(* PLC project Recipe_Tool, Beckhoff Automation GmbH TwinCAT PLC Control 3.5.3.40 *)
(* stored: creationDateTime 2014-11-22T03:13:17.8029505, modificationDateTime 2014-11-22T03:13:17.8029505 *)

FUNCTION_BLOCK Recipe_10051_FreePassion
  VAR_INPUT
    execute : BOOL;
    Order : DUT_RECIPEORDER;
  END_VAR
  VAR_OUTPUT
    RecipeInfo : DUT_RECIPEOFFER;
    RecipeDone : BOOL;
    InitDone : BOOL;
  END_VAR
  VAR
    userparametersum : LREAL;
    StepDone : BOOL;
    i : INT;
  END_VAR

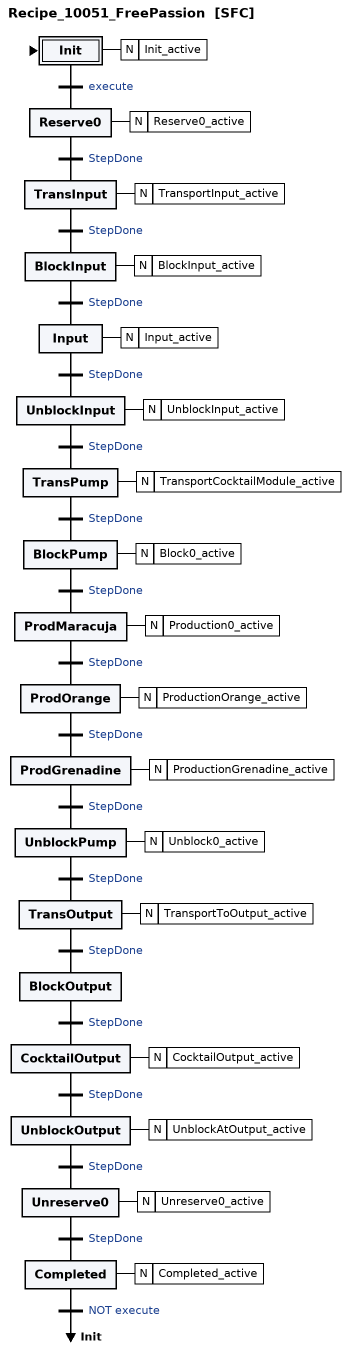
INITIAL_STEP Init:
  Init_active(N);
END_STEP
TRANSITION FROM Init TO Reserve0
  := execute;
END_TRANSITION
STEP Reserve0:
  Reserve0_active(N);
END_STEP
TRANSITION FROM Reserve0 TO TransInput
  := StepDone;
END_TRANSITION
STEP TransInput:
  TransportInput_active(N);
END_STEP
TRANSITION FROM TransInput TO BlockInput
  := StepDone;
END_TRANSITION
STEP BlockInput:
  BlockInput_active(N);
END_STEP
TRANSITION FROM BlockInput TO Input
  := StepDone;
END_TRANSITION
STEP Input:
  Input_active(N);
END_STEP
TRANSITION FROM Input TO UnblockInput
  := StepDone;
END_TRANSITION
STEP UnblockInput:
  UnblockInput_active(N);
END_STEP
TRANSITION FROM UnblockInput TO TransPump
  := StepDone;
END_TRANSITION
STEP TransPump:
  TransportCocktailModule_active(N);
END_STEP
TRANSITION FROM TransPump TO BlockPump
  := StepDone;
END_TRANSITION
STEP BlockPump:
  Block0_active(N);
END_STEP
TRANSITION FROM BlockPump TO ProdMaracuja
  := StepDone;
END_TRANSITION
STEP ProdMaracuja:
  Production0_active(N);
END_STEP
TRANSITION FROM ProdMaracuja TO ProdOrange
  := StepDone;
END_TRANSITION
STEP ProdOrange:
  ProductionOrange_active(N);
END_STEP
TRANSITION FROM ProdOrange TO ProdGrenadine
  := StepDone;
END_TRANSITION
STEP ProdGrenadine:
  ProductionGrenadine_active(N);
END_STEP
TRANSITION FROM ProdGrenadine TO UnblockPump
  := StepDone;
END_TRANSITION
STEP UnblockPump:
  Unblock0_active(N);
END_STEP
TRANSITION FROM UnblockPump TO TransOutput
  := StepDone;
END_TRANSITION
STEP TransOutput:
  TransportToOutput_active(N);
END_STEP
TRANSITION FROM TransOutput TO BlockOutput
  := StepDone;
END_TRANSITION
STEP BlockOutput:
END_STEP
TRANSITION FROM BlockOutput TO CocktailOutput
  := StepDone;
END_TRANSITION
STEP CocktailOutput:
  CocktailOutput_active(N);
END_STEP
TRANSITION FROM CocktailOutput TO UnblockOutput
  := StepDone;
END_TRANSITION
STEP UnblockOutput:
  UnblockAtOutput_active(N);
END_STEP
TRANSITION FROM UnblockOutput TO Unreserve0
  := StepDone;
END_TRANSITION
STEP Unreserve0:
  Unreserve0_active(N);
END_STEP
TRANSITION FROM Unreserve0 TO Completed
  := StepDone;
END_TRANSITION
STEP Completed:
  Completed_active(N);
END_STEP
TRANSITION FROM Completed TO Init
  := NOT execute;
END_TRANSITION

ACTION Completed_active:
                RecipeDone := TRUE;
StepDone := FALSE;
              
END_ACTION

ACTION Init_active:
                RecipeDone := FALSE;

// Initialisation of Recipe Parameters an name etc
RecipeInfo.Name := 'Free Passion';
RecipeInfo.Description := 'Sweet cocktail combining the sourness of Maracuja juice with the sweetness of grenadine syrup';
RecipeInfo.Dummy := FALSE;
RecipeInfo.RecipeID := 10051; 	// 
Initdone := TRUE;

//Parameter 0:

	RecipeInfo.UserParameter[0].Dummy 		:= FALSE
	RecipeInfo.UserParameter[0].Default		:= '200'
	RecipeInfo.UserParameter[0].Description	:= 'Gives the total fluid amount in the glass'
	RecipeInfo.UserParameter[0].MaxValue	:= 200
	RecipeInfo.UserParameter[0].MinValue	:= 10
	RecipeInfo.UserParameter[0].Name		:= 'Amount'
	RecipeInfo.UserParameter[0].Unit		:= 'ml'
	
//Parameter 1:

	RecipeInfo.UserParameter[1].Dummy 		:= FALSE
	RecipeInfo.UserParameter[1].Default		:= '50'
	RecipeInfo.UserParameter[1].Description	:= 'Maracuja Juice'
	RecipeInfo.UserParameter[1].MaxValue	:= 100
	RecipeInfo.UserParameter[1].MinValue	:= 1
	RecipeInfo.UserParameter[1].Name		:= 'Maracuja Juice'
	RecipeInfo.UserParameter[1].Unit		:= 'ml'
	
//Parameter 2:

	RecipeInfo.UserParameter[2].Dummy 		:= FALSE
	RecipeInfo.UserParameter[2].Default		:= '35'
	RecipeInfo.UserParameter[2].Description	:= 'Orange Juice'
	RecipeInfo.UserParameter[2].MaxValue	:= 100
	RecipeInfo.UserParameter[2].MinValue	:= 1
	RecipeInfo.UserParameter[2].Name		:= 'Orange Juice'
	RecipeInfo.UserParameter[2].Unit		:= 'ml'

//Parameter 3:

	RecipeInfo.UserParameter[3].Dummy 		:= FALSE
	RecipeInfo.UserParameter[3].Default		:= '15'
	RecipeInfo.UserParameter[3].Description	:= 'Grenadine Syrup'
	RecipeInfo.UserParameter[3].MaxValue	:= 50
	RecipeInfo.UserParameter[3].MinValue	:= 1
	RecipeInfo.UserParameter[3].Name		:= 'Grenadine Syrup'
	RecipeInfo.UserParameter[3].Unit		:= 'ml'
	
	
	
//Parameter 1:
(*
	RecipeInfo.UserParameter[1].Dummy 		:= 
	RecipeInfo.UserParameter[1].Default		:=
	RecipeInfo.UserParameter[1].Description	:=
	RecipeInfo.UserParameter[1].MaxValue	:=
	RecipeInfo.UserParameter[1].MinValue	:=
	RecipeInfo.UserParameter[1].Name		:=
	RecipeInfo.UserParameter[1].Unit		:=
*)
//Parameter 2:

(*
	RecipeInfo.UserParameter[2].Dummy 		:= 
	RecipeInfo.UserParameter[2].Default		:=
	RecipeInfo.UserParameter[2].Description	:=
	RecipeInfo.UserParameter[2].MaxValue	:=
	RecipeInfo.UserParameter[2].MinValue	:=
	RecipeInfo.UserParameter[2].Name		:=
	RecipeInfo.UserParameter[2].Unit		:=
*)

//Parameter 3:

(*
	RecipeInfo.UserParameter[3].Dummy 		:= 
	RecipeInfo.UserParameter[3].Default		:=
	RecipeInfo.UserParameter[3].Description	:=
	RecipeInfo.UserParameter[3].MaxValue	:=
	RecipeInfo.UserParameter[3].MinValue	:=
	RecipeInfo.UserParameter[3].Name		:=
	RecipeInfo.UserParameter[3].Unit		:=
*)

//Parameter 4:

(*
	RecipeInfo.UserParameter[4].Dummy 		:= 
	RecipeInfo.UserParameter[4].Default		:=
	RecipeInfo.UserParameter[4].Description	:=
	RecipeInfo.UserParameter[4].MaxValue	:=
	RecipeInfo.UserParameter[4].MinValue	:=
	RecipeInfo.UserParameter[4].Name		:=
	RecipeInfo.UserParameter[4].Unit		:=
*)


//Parameter 5:

(*
	RecipeInfo.UserParameter[5].Dummy 		:= 
	RecipeInfo.UserParameter[5].Default		:=
	RecipeInfo.UserParameter[5].Description	:=
	RecipeInfo.UserParameter[5].MaxValue	:=
	RecipeInfo.UserParameter[5].MinValue	:=
	RecipeInfo.UserParameter[5].Name		:=
	RecipeInfo.UserParameter[5].Unit		:=
*)
              
END_ACTION

ACTION Reserve0_active:
                StepDone := FALSE;
RecipeDone := FALSE;
//Skill auswählen
ExecuteSkill.SkillID 		:= 1310;
ExecuteSkill.SkillName	 	:= 'Reserve';

//Parameter setzen

ExecuteSkill.Parameter[1].ID := 1;
ExecuteSkill.Parameter[1].Name := 'TaskID';
ExecuteSkill.Parameter[1].Value := Order.TaskID;


(*
ExecuteSkill.Parameter[2].ID := ;
ExecuteSkill.Parameter[2].Name := '';
ExecuteSkill.Parameter[2].Value := ;
*)

(*
ExecuteSkill.Parameter[3].ID := ;
ExecuteSkill.Parameter[3].Name := '';
ExecuteSkill.Parameter[3].Value := ;
*)

(*
ExecuteSkill.Parameter[4].ID := ;
ExecuteSkill.Parameter[4].Name := '';
ExecuteSkill.Parameter[4].Value := ;
*)

(*
ExecuteSkill.Parameter[5].ID := ;
ExecuteSkill.Parameter[5].Name := '';
ExecuteSkill.Parameter[5].Value := ;
*)



ExecuteSkill();

StepDone := ExecuteSkill.Done;
              
END_ACTION

ACTION Production0_active:
                StepDone := FALSE;

userparametersum := 0;
FOR i := 1 TO UserParameterCnt DO
	IF NOT order.UserParameter[i].Value = 0 THEN
		userparametersum := userparametersum + order.UserParameter[i].Value;
	END_IF
END_FOR
//Skill auswählen
ExecuteSkill.SkillID 		:= 1113;
ExecuteSkill.SkillName	 	:= 'Marajuca Juice';

//Parameter setzen

ExecuteSkill.Parameter[1].ID := 1;
ExecuteSkill.Parameter[1].Name := 'Quantity';
//order.userParameter[0] = amount
ExecuteSkill.Parameter[1].Value := order.UserParameter[0].Value * order.UserParameter[0].Value / userparametersum;//Summe aller Zutatenmengen;


(*
ExecuteSkill.Parameter[2].ID := ;
ExecuteSkill.Parameter[2].Name := '';
ExecuteSkill.Parameter[2].Value := ;
*)

(*
ExecuteSkill.Parameter[3].ID := ;
ExecuteSkill.Parameter[3].Name := '';
ExecuteSkill.Parameter[3].Value := ;
*)

(*
ExecuteSkill.Parameter[4].ID := ;
ExecuteSkill.Parameter[4].Name := '';
ExecuteSkill.Parameter[4].Value := ;
*)

(*
ExecuteSkill.Parameter[5].ID := ;
ExecuteSkill.Parameter[5].Name := '';
ExecuteSkill.Parameter[5].Value := ;
*)



ExecuteSkill();

StepDone := ExecuteSkill.Done;
              
END_ACTION

ACTION ProductionOrange_active:
                StepDone := FALSE;

//Skill auswählen
ExecuteSkill.SkillID 		:= 1117;
ExecuteSkill.SkillName	 	:= 'Orange';

//Parameter setzen

ExecuteSkill.Parameter[1].ID := 1;
ExecuteSkill.Parameter[1].Name := 'Quantity';
//order.userParameter[0] = amount
ExecuteSkill.Parameter[1].Value := order.UserParameter[0].Value * order.UserParameter[1].Value / userparametersum;//Summe aller Zutatenmengen;



(*
ExecuteSkill.Parameter[2].ID := ;
ExecuteSkill.Parameter[2].Name := '';
ExecuteSkill.Parameter[2].Value := ;
*)

(*
ExecuteSkill.Parameter[3].ID := ;
ExecuteSkill.Parameter[3].Name := '';
ExecuteSkill.Parameter[3].Value := ;
*)

(*
ExecuteSkill.Parameter[4].ID := ;
ExecuteSkill.Parameter[4].Name := '';
ExecuteSkill.Parameter[4].Value := ;
*)

(*
ExecuteSkill.Parameter[5].ID := ;
ExecuteSkill.Parameter[5].Name := '';
ExecuteSkill.Parameter[5].Value := ;
*)



ExecuteSkill();

StepDone := ExecuteSkill.Done;
              
END_ACTION

ACTION ProductionGrenadine_active:
                StepDone := FALSE;

//Skill auswählen
ExecuteSkill.SkillID 		:= 1111;
ExecuteSkill.SkillName	 	:= 'Grenadine';

//Parameter setzen

ExecuteSkill.Parameter[1].ID := 1;
ExecuteSkill.Parameter[1].Name := 'Quantity';
//order.userParameter[0] = amount
ExecuteSkill.Parameter[1].Value := order.UserParameter[0].Value * order.UserParameter[2].Value / userparametersum; //Summe aller Zutatenmengen;



(*
ExecuteSkill.Parameter[2].ID := ;
ExecuteSkill.Parameter[2].Name := '';
ExecuteSkill.Parameter[2].Value := ;
*)

(*
ExecuteSkill.Parameter[3].ID := ;
ExecuteSkill.Parameter[3].Name := '';
ExecuteSkill.Parameter[3].Value := ;
*)

(*
ExecuteSkill.Parameter[4].ID := ;
ExecuteSkill.Parameter[4].Name := '';
ExecuteSkill.Parameter[4].Value := ;
*)

(*
ExecuteSkill.Parameter[5].ID := ;
ExecuteSkill.Parameter[5].Name := '';
ExecuteSkill.Parameter[5].Value := ;
*)



ExecuteSkill();

StepDone := ExecuteSkill.Done;
              
END_ACTION

ACTION TransportCocktailModule_active:
                StepDone := FALSE;

//Skill auswählen
ExecuteSkill.SkillID 		:= 1320;
ExecuteSkill.SkillName	 	:= 'Transport';

//Parameter setzen

ExecuteSkill.Parameter[3].ID := 3;
ExecuteSkill.Parameter[3].Name := 'Velocity';
ExecuteSkill.Parameter[3].Value := 300;



ExecuteSkill.Parameter[1].ID :=  1;
ExecuteSkill.Parameter[1].Name := 'TargetPosition X';
ExecuteSkill.Parameter[1].Value := 30 ;
ExecuteSkill.Parameter[1].StringValue := '#DP#2#XPosition';



ExecuteSkill.Parameter[2].ID := 2;
ExecuteSkill.Parameter[2].Name := 'TargetPosition Z';
ExecuteSkill.Parameter[2].Value := 10;// ZCookieModule - ZCookieModuleCalibration - 2* Cookiethickness + toppingthickness+ Preasureheight  ;



(*
ExecuteSkill.Parameter[4].ID := 4;
ExecuteSkill.Parameter[4].Name := 'Acceleration';
ExecuteSkill.Parameter[4].Value := 0 ;
*)

(*
ExecuteSkill.Parameter[5].ID := ;
ExecuteSkill.Parameter[5].Name := '';
ExecuteSkill.Parameter[5].Value := ;
*)



ExecuteSkill();

StepDone := ExecuteSkill.Done;
              
END_ACTION

ACTION Block0_active:
                StepDone := FALSE;

//Skill auswählen
ExecuteSkill.SkillID 		:= 1315;
ExecuteSkill.SkillName	 	:= 'Block';

//Parameter setzen

ExecuteSkill.Parameter[1].ID := 1;
ExecuteSkill.Parameter[1].Name := 'TaskID';
ExecuteSkill.Parameter[1].Value := Order.TaskID;


(*
ExecuteSkill.Parameter[2].ID := ;
ExecuteSkill.Parameter[2].Name := '';
ExecuteSkill.Parameter[2].Value := ;
*)

(*
ExecuteSkill.Parameter[3].ID := ;
ExecuteSkill.Parameter[3].Name := '';
ExecuteSkill.Parameter[3].Value := ;
*)

(*
ExecuteSkill.Parameter[4].ID := ;
ExecuteSkill.Parameter[4].Name := '';
ExecuteSkill.Parameter[4].Value := ;
*)

(*
ExecuteSkill.Parameter[5].ID := ;
ExecuteSkill.Parameter[5].Name := '';
ExecuteSkill.Parameter[5].Value := ;
*)



ExecuteSkill();

StepDone := ExecuteSkill.Done;
              
END_ACTION

ACTION Unblock0_active:
                StepDone := FALSE;

//Skill auswählen
ExecuteSkill.SkillID 		:= 1316;
ExecuteSkill.SkillName	 	:= 'Unblock';

//Parameter setzen

ExecuteSkill.Parameter[1].ID := 1;
ExecuteSkill.Parameter[1].Name := 'TaskID';
ExecuteSkill.Parameter[1].Value := Order.TaskID;


(*
ExecuteSkill.Parameter[2].ID := ;
ExecuteSkill.Parameter[2].Name := '';
ExecuteSkill.Parameter[2].Value := ;
*)

(*
ExecuteSkill.Parameter[3].ID := ;
ExecuteSkill.Parameter[3].Name := '';
ExecuteSkill.Parameter[3].Value := ;
*)

(*
ExecuteSkill.Parameter[4].ID := ;
ExecuteSkill.Parameter[4].Name := '';
ExecuteSkill.Parameter[4].Value := ;
*)

(*
ExecuteSkill.Parameter[5].ID := ;
ExecuteSkill.Parameter[5].Name := '';
ExecuteSkill.Parameter[5].Value := ;
*)



ExecuteSkill();

StepDone := ExecuteSkill.Done;
              
END_ACTION

ACTION TransportToOutput_active:
                StepDone := FALSE;

//Skill auswählen
ExecuteSkill.SkillID 		:= 1320;
ExecuteSkill.SkillName	 	:= 'Transport';

//Parameter setzen

ExecuteSkill.Parameter[3].ID := 3;
ExecuteSkill.Parameter[3].Name := 'Velocity';
ExecuteSkill.Parameter[3].Value := 300;



ExecuteSkill.Parameter[1].ID :=  1;
ExecuteSkill.Parameter[1].Name := 'TargetPosition X';
ExecuteSkill.Parameter[1].Value := 30 ;
ExecuteSkill.Parameter[1].StringValue := '';



ExecuteSkill.Parameter[2].ID := 2;
ExecuteSkill.Parameter[2].Name := 'TargetPosition Z';
ExecuteSkill.Parameter[2].Value := 90;// ZCookieModule - ZCookieModuleCalibration - 2* Cookiethickness + toppingthickness+ Preasureheight  ;



(* ExecuteSkill.Parameter[4].ID := 4;
ExecuteSkill.Parameter[4].Name := 'Acceleration';
ExecuteSkill.Parameter[4].Value :=0 ;

*)
(*
ExecuteSkill.Parameter[5].ID := ;
ExecuteSkill.Parameter[5].Name := '';
ExecuteSkill.Parameter[5].Value := ;
*)



ExecuteSkill();

StepDone := ExecuteSkill.Done;
              
END_ACTION

ACTION CocktailOutput_active:
                StepDone := FALSE;

//Skill auswählen
ExecuteSkill.SkillID 		:= 1403;
ExecuteSkill.SkillName	 	:= 'Output';

//Parameter setzen

ExecuteSkill.Parameter[1].ID := 1;
ExecuteSkill.Parameter[1].Name := 'TaskID';
ExecuteSkill.Parameter[1].Value := Order.TaskID;


(*
ExecuteSkill.Parameter[2].ID := ;
ExecuteSkill.Parameter[2].Name := '';
ExecuteSkill.Parameter[2].Value := ;
*)

(*
ExecuteSkill.Parameter[3].ID := ;
ExecuteSkill.Parameter[3].Name := '';
ExecuteSkill.Parameter[3].Value := ;
*)

(*
ExecuteSkill.Parameter[4].ID := ;
ExecuteSkill.Parameter[4].Name := '';
ExecuteSkill.Parameter[4].Value := ;
*)

(*
ExecuteSkill.Parameter[5].ID := ;
ExecuteSkill.Parameter[5].Name := '';
ExecuteSkill.Parameter[5].Value := ;
*)



ExecuteSkill();

StepDone := ExecuteSkill.Done;
              
END_ACTION

ACTION UnblockAtOutput_active:
                StepDone := FALSE;

//Skill auswählen
ExecuteSkill.SkillID 		:= 1316;
ExecuteSkill.SkillName	 	:= 'Unblock';

//Parameter setzen

ExecuteSkill.Parameter[1].ID := 1;
ExecuteSkill.Parameter[1].Name := 'TaskID';
ExecuteSkill.Parameter[1].Value := Order.TaskID;


(*
ExecuteSkill.Parameter[2].ID := ;
ExecuteSkill.Parameter[2].Name := '';
ExecuteSkill.Parameter[2].Value := ;
*)

(*
ExecuteSkill.Parameter[3].ID := ;
ExecuteSkill.Parameter[3].Name := '';
ExecuteSkill.Parameter[3].Value := ;
*)

(*
ExecuteSkill.Parameter[4].ID := ;
ExecuteSkill.Parameter[4].Name := '';
ExecuteSkill.Parameter[4].Value := ;
*)

(*
ExecuteSkill.Parameter[5].ID := ;
ExecuteSkill.Parameter[5].Name := '';
ExecuteSkill.Parameter[5].Value := ;
*)



ExecuteSkill();

StepDone := ExecuteSkill.Done;
              
END_ACTION

ACTION Unreserve0_active:
                StepDone := FALSE;

//Skill auswählen
ExecuteSkill.SkillID 		:= 1311;
ExecuteSkill.SkillName	 	:= 'Unreserve';

//Parameter setzen

ExecuteSkill.Parameter[1].ID := 1;
ExecuteSkill.Parameter[1].Name := 'TaskID';
ExecuteSkill.Parameter[1].Value := Order.TaskID;


(*
ExecuteSkill.Parameter[2].ID := ;
ExecuteSkill.Parameter[2].Name := '';
ExecuteSkill.Parameter[2].Val ue := ;
*)

(*
ExecuteSkill.Parameter[3].ID := ;
ExecuteSkill.Parameter[3].Name := '';
ExecuteSkill.Parameter[3].Value := ;
*)

(*
ExecuteSkill.Parameter[4].ID := ;
ExecuteSkill.Parameter[4].Name := '';
ExecuteSkill.Parameter[4].Value := ;
*)

(*
ExecuteSkill.Parameter[5].ID := ;
ExecuteSkill.Parameter[5].Name := '';
ExecuteSkill.Parameter[5].Value := ;
*)



ExecuteSkill();

StepDone := ExecuteSkill.Done;
              
END_ACTION

ACTION TransportInput_active:
                StepDone := FALSE;

//Skill auswählen
ExecuteSkill.SkillID 		:= 1320;
ExecuteSkill.SkillName	 	:= 'Transport';

//Parameter setzen

ExecuteSkill.Parameter[3].ID := 3;
ExecuteSkill.Parameter[3].Name := 'Velocity';
ExecuteSkill.Parameter[3].Value := 300;



ExecuteSkill.Parameter[1].ID :=  1;
ExecuteSkill.Parameter[1].Name := 'TargetPosition X';
ExecuteSkill.Parameter[1].Value := 30 ;
ExecuteSkill.Parameter[1].StringValue := '#DP#2#XPosition';



ExecuteSkill.Parameter[2].ID := 2;
ExecuteSkill.Parameter[2].Name := 'TargetPosition Z';
ExecuteSkill.Parameter[2].Value := 10;// ZCookieModule - ZCookieModuleCalibration - 2* Cookiethickness + toppingthickness+ Preasureheight  ;



(*
ExecuteSkill.Parameter[4].ID := 4;
ExecuteSkill.Parameter[4].Name := 'Acceleration';
ExecuteSkill.Parameter[4].Value := 0 ;
*)

(*
ExecuteSkill.Parameter[5].ID := ;
ExecuteSkill.Parameter[5].Name := '';
ExecuteSkill.Parameter[5].Value := ;
*)



ExecuteSkill();

StepDone := ExecuteSkill.Done;
              
END_ACTION

ACTION BlockInput_active:
                StepDone := FALSE;

//Skill auswählen
ExecuteSkill.SkillID 		:= 1315;
ExecuteSkill.SkillName	 	:= 'Block';

//Parameter setzen

ExecuteSkill.Parameter[1].ID := 1;
ExecuteSkill.Parameter[1].Name := 'TaskID';
ExecuteSkill.Parameter[1].Value := Order.TaskID;


(*
ExecuteSkill.Parameter[2].ID := ;
ExecuteSkill.Parameter[2].Name := '';
ExecuteSkill.Parameter[2].Value := ;
*)

(*
ExecuteSkill.Parameter[3].ID := ;
ExecuteSkill.Parameter[3].Name := '';
ExecuteSkill.Parameter[3].Value := ;
*)

(*
ExecuteSkill.Parameter[4].ID := ;
ExecuteSkill.Parameter[4].Name := '';
ExecuteSkill.Parameter[4].Value := ;
*)

(*
ExecuteSkill.Parameter[5].ID := ;
ExecuteSkill.Parameter[5].Name := '';
ExecuteSkill.Parameter[5].Value := ;
*)



ExecuteSkill();

StepDone := ExecuteSkill.Done;
              
END_ACTION

ACTION Input_active:
                StepDone := FALSE;

//Skill auswählen
ExecuteSkill.SkillID 		:= 1402;
ExecuteSkill.SkillName	 	:= 'Input';

//Parameter setzen

ExecuteSkill.Parameter[1].ID := 1;
ExecuteSkill.Parameter[1].Name := 'TaskID';
ExecuteSkill.Parameter[1].Value := Order.TaskID;


(*
ExecuteSkill.Parameter[2].ID := ;
ExecuteSkill.Parameter[2].Name := '';
ExecuteSkill.Parameter[2].Value := ;
*)

(*
ExecuteSkill.Parameter[3].ID := ;
ExecuteSkill.Parameter[3].Name := '';
ExecuteSkill.Parameter[3].Value := ;
*)

(*
ExecuteSkill.Parameter[4].ID := ;
ExecuteSkill.Parameter[4].Name := '';
ExecuteSkill.Parameter[4].Value := ;
*)

(*
ExecuteSkill.Parameter[5].ID := ;
ExecuteSkill.Parameter[5].Name := '';
ExecuteSkill.Parameter[5].Value := ;
*)



ExecuteSkill();

StepDone := ExecuteSkill.Done;
              
END_ACTION

ACTION UnblockInput_active:
                StepDone := FALSE;

//Skill auswählen
ExecuteSkill.SkillID 		:= 1316;
ExecuteSkill.SkillName	 	:= 'Unblock';

//Parameter setzen

ExecuteSkill.Parameter[1].ID := 1;
ExecuteSkill.Parameter[1].Name := 'TaskID';
ExecuteSkill.Parameter[1].Value := Order.TaskID;


(*
ExecuteSkill.Parameter[2].ID := ;
ExecuteSkill.Parameter[2].Name := '';
ExecuteSkill.Parameter[2].Value := ;
*)

(*
ExecuteSkill.Parameter[3].ID := ;
ExecuteSkill.Parameter[3].Name := '';
ExecuteSkill.Parameter[3].Value := ;
*)

(*
ExecuteSkill.Parameter[4].ID := ;
ExecuteSkill.Parameter[4].Name := '';
ExecuteSkill.Parameter[4].Value := ;
*)

(*
ExecuteSkill.Parameter[5].ID := ;
ExecuteSkill.Parameter[5].Name := '';
ExecuteSkill.Parameter[5].Value := ;
*)



ExecuteSkill();

StepDone := ExecuteSkill.Done;
              
END_ACTION
END_FUNCTION_BLOCK
